{attribute 'strict'}
TYPE E_CognexCameraGetValueEasyBuilderStatus :
(
	WAITING_FOR_STATUS_CODE						:= 2,
	THE_COMMAND_WAS_EXECUTED_SUCCESSFULLY		:= 1,
	UNRECOGNIZED_COMMAND 						:= 0,
	THE_SYMBOLIC_TAG_IS_INVALID					:= -1,
	THE_COMMAND_COULD_NOT_BE_EXECUTED 			:= -2
);
END_TYPE

(* stored: Version 1.1.0.1, ProductVersion 3.1.4024.9
   DUT E_CognexCameraGetValueEasyBuilderStatus: Id {dda778ae-a76e-4f34-9038-abade2409639} *)
